// TIA Portal project "Prakticne-3_sabirac" (V16)

(* hardware
DEVICE "S7-1200 station_1"  S7-1200 Station
   slot 0: "Rack_0"  S7-1200 Rack  Rack  V1.0
   slot 1: "PLC_1"  CPU 1214C AC/DC/Rly  6ES7 214-1BG31-0XB0  V3.0
*)

// ===== PLC "PLC_1"  CPU 1214C AC/DC/Rly =====

VAR_GLOBAL   // PLC tag table "Default tag table"
   "Clock_Byte" AT %MB10 : Byte;
   "Clock_10Hz" AT %M10.0 : Bool;
   "Clock_5Hz" AT %M10.1 : Bool;
   "Clock_2.5Hz" AT %M10.2 : Bool;
   "Clock_2Hz" AT %M10.3 : Bool;
   "Clock_1.25Hz" AT %M10.4 : Bool;
   "Clock_1Hz" AT %M10.5 : Bool;
   "Clock_0.625Hz" AT %M10.6 : Bool;
   "Clock_0.5Hz" AT %M10.7 : Bool;
   "Tag_1" AT %M20.0 : Bool;
   "Tag_2" AT %M20.1 : Bool;
   "Tag_3" AT %M20.2 : Bool;
   "Tag_4" AT %M20.3 : Bool;
END_VAR

VAR_GLOBAL   // PLC tag table "Tag table_1"
   "Prekidac 1" AT %I0.0 : Bool;
   "Prekidac 2" AT %I0.1 : Bool;
   "Prekidac 3" AT %I0.2 : Bool;
   "Prekidac 4" AT %I0.3 : Bool;
   "Prekidac 5" AT %I0.4 : Bool;
   "Prekidac 6" AT %I0.5 : Bool;
   "Prekidac 7" AT %I0.6 : Bool;
   "Induktivni senzor" AT %I1.0 : Bool;
   "Pun krig napravljen" AT %I1.1 : Bool;
   "Dioda 2" AT %Q0.0 : Bool;
   "Dioda 3" AT %Q0.1 : Bool;
   "Dioda 4" AT %Q0.2 : Bool;
   "Dioda 5" AT %Q0.3 : Bool;
   "Motor suprotno od kazaljke" AT %Q0.4 : Bool;
   "Motor u smeru kazaljke" AT %Q0.5 : Bool;
END_VAR

DATA_BLOCK "DB_memorija_sabiraca"   // DB2
{ S7_Optimized_Access := 'TRUE' }
VERSION : 0.1
   VAR
      broj_prolaza : Int := 3;
   END_VAR
BEGIN
END_DATA_BLOCK

FUNCTION "FC_kretanje" : Void   // FC1, LAD
{ S7_Optimized_Access := 'TRUE' }
VERSION : 0.1
   VAR_TEMP   // added for the SCL form of the ladder/FBD networks
      _w1 : Bool;
   END_VAR
BEGIN

REGION Network 1
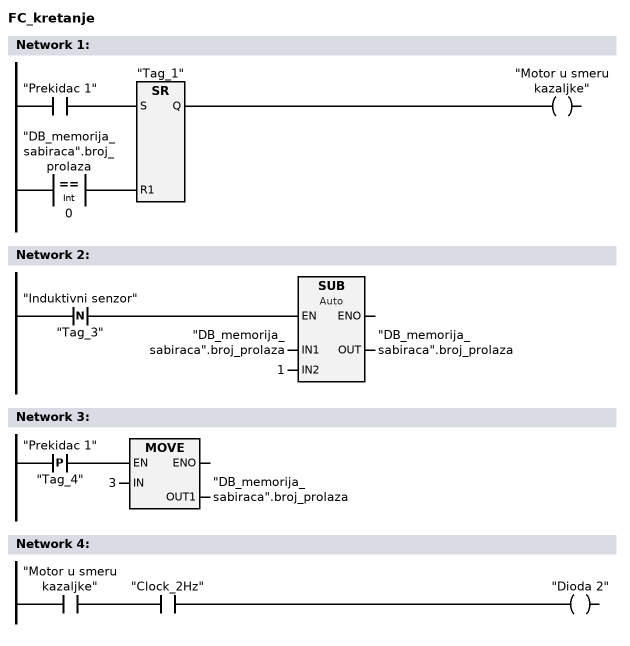
   RUNG wire#powerrail
      Contact( "Prekidac 1" )
      S_SR(operand := "Tag_1", r1 := wire#w1)
      Coil( "Motor u smeru kazaljke" )
   END_RUNG
   RUNG wire#powerrail
      { S7_Templates := "SrcType := Int" } EQ_Contact(in1 := "DB_memorija_sabiraca".broj_prolaza, in2 := 0)
   END_RUNG wire#w1
   // the same network as SCL:
   IF "Prekidac 1" THEN
       "Tag_1" := TRUE;   // SR flip-flop
   END_IF;
   IF "DB_memorija_sabiraca".broj_prolaza = 0 THEN "Tag_1" := FALSE; END_IF;
   "Motor u smeru kazaljke" := "Tag_1";
END_REGION

REGION Network 2
   RUNG wire#powerrail
      N_Contact(operand := "Induktivni senzor", bit := "Tag_3")
      { S7_GenerateENO := "TRUE" } Sub(in1 := "DB_memorija_sabiraca".broj_prolaza, in2 := 1, out => "DB_memorija_sabiraca".broj_prolaza)
   END_RUNG
   // the same network as SCL:
   #_w1 := NOT "Induktivni senzor" AND "Tag_3";   // falling edge of "Induktivni senzor"
   "Tag_3" := "Induktivni senzor";
   IF #_w1 THEN "DB_memorija_sabiraca".broj_prolaza := "DB_memorija_sabiraca".broj_prolaza - 1; END_IF;
END_REGION

REGION Network 3
   RUNG wire#powerrail
      P_Contact(operand := "Prekidac 1", bit := "Tag_4")
      { S7_GenerateENO := "TRUE" } Move(in := 3, out1 => "DB_memorija_sabiraca".broj_prolaza)
   END_RUNG
   // the same network as SCL:
   #_w1 := "Prekidac 1" AND NOT "Tag_4";   // rising edge of "Prekidac 1"
   "Tag_4" := "Prekidac 1";
   IF #_w1 THEN "DB_memorija_sabiraca".broj_prolaza := 3; END_IF;
END_REGION

REGION Network 4
   RUNG wire#powerrail
      Contact( "Motor u smeru kazaljke" )
      Contact( "Clock_2Hz" )
      Coil( "Dioda 2" )
   END_RUNG
   // the same network as SCL:
   "Dioda 2" := "Motor u smeru kazaljke" AND "Clock_2Hz";
END_REGION
END_FUNCTION

ORGANIZATION_BLOCK "Main"   // OB1, LAD, ProgramCycle
TITLE = "Main Program Sweep (Cycle)"
{ S7_Optimized_Access := 'TRUE' }
VERSION : 0.1
BEGIN

REGION Network 1
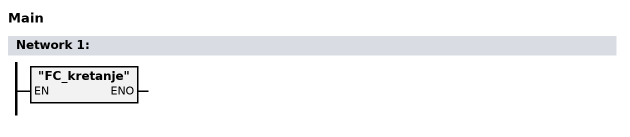
   RUNG wire#powerrail
      "FC_kretanje"()
   END_RUNG
   // the same network as SCL:
   "FC_kretanje"();
END_REGION
END_ORGANIZATION_BLOCK